// Mitsubishi GX Works2 project: 8   PLC: FX3U/FX3UC

// task Task_01 (event TRUE, interval 0, priority 31): POU_01

PROGRAM POU_01
VAR
  wstep : INT;
END_VAR
IF M8002 THEN
	wstep := 0;
END_IF;

CASE wstep OF
	0:
	IF M40 THEN
		wstep := 20;
	END_IF;
	
	20:
	Y0 := FALSE;
	
	IF M45 THEN
		wstep := 21;
	END_IF;

	IF M46 THEN
		wstep := 22;
	END_IF;
	
	21:
	Y1 := TRUE;
	
	IF M42 THEN
		wstep := 30;
	END_IF;
	
	22:
	Y1 := TRUE;
	
	IF M43 THEN
		wstep := 40;
	END_IF;
	
	30:
	Y0 := FALSE;
	Y1 := FALSE;
	
	IF M44 THEN
		wstep := 31;
	END_IF;
	
	IF M46 THEN
		wstep := 32;
	END_IF;
	
	31:
	Y0 := TRUE;
	
	IF M41 THEN
		wstep := 20;
	END_IF;
	
	32:
	Y1 := TRUE;
	
	IF M43 THEN
		wstep := 40;
	END_IF;
	
	40:
	Y1 := FALSE;
	
	IF M44 THEN
		wstep  := 41;
	END_IF;
	
	IF M45 THEN
		wstep := 42;
	END_IF;
	
	41:
	Y0 := TRUE;
	
	IF M41 THEN
		wstep := 20;
	END_IF;
	
	42:
	Y0 := TRUE;
	
	IF M42 THEN
		wstep := 30;
	END_IF;

END_CASE;
END_PROGRAM
